PROGRAM MAIN
VAR
	fSin		: REAL;
	fTheta		: REAL := -3.14;
	fbSampling	: TON;
END_VAR

fbSampling(In:=TRUE, PT:=T#1S);

IF fbSampling.Q THEN
	IF fTheta >= 3.14 THEN
		fTheta := -3.14;
	END_IF
	fSin := SIN(fTheta);
	fTheta := fTheta + 0.01;
	fbSampling(In:=FALSE);
END_IF

END_PROGRAM

(* stored: Version 1.1.0.1, ProductVersion 3.1.4024.9
   POU MAIN: Id {fbf1a1d8-33d2-4178-84e1-36bef6184fbb}, SpecialFunc None *)
